PROGRAM GL9_Conveyor
VAR
	
	RUN_FWD_BIT_TO_EXIT : BOOL; // RUN FORWARD TO EXIT POSITION AFTER DROP
END_VAR
VAR // added by the converter: edge detectors and wires of the graphical bodies
    _w1 : BOOL;
END_VAR

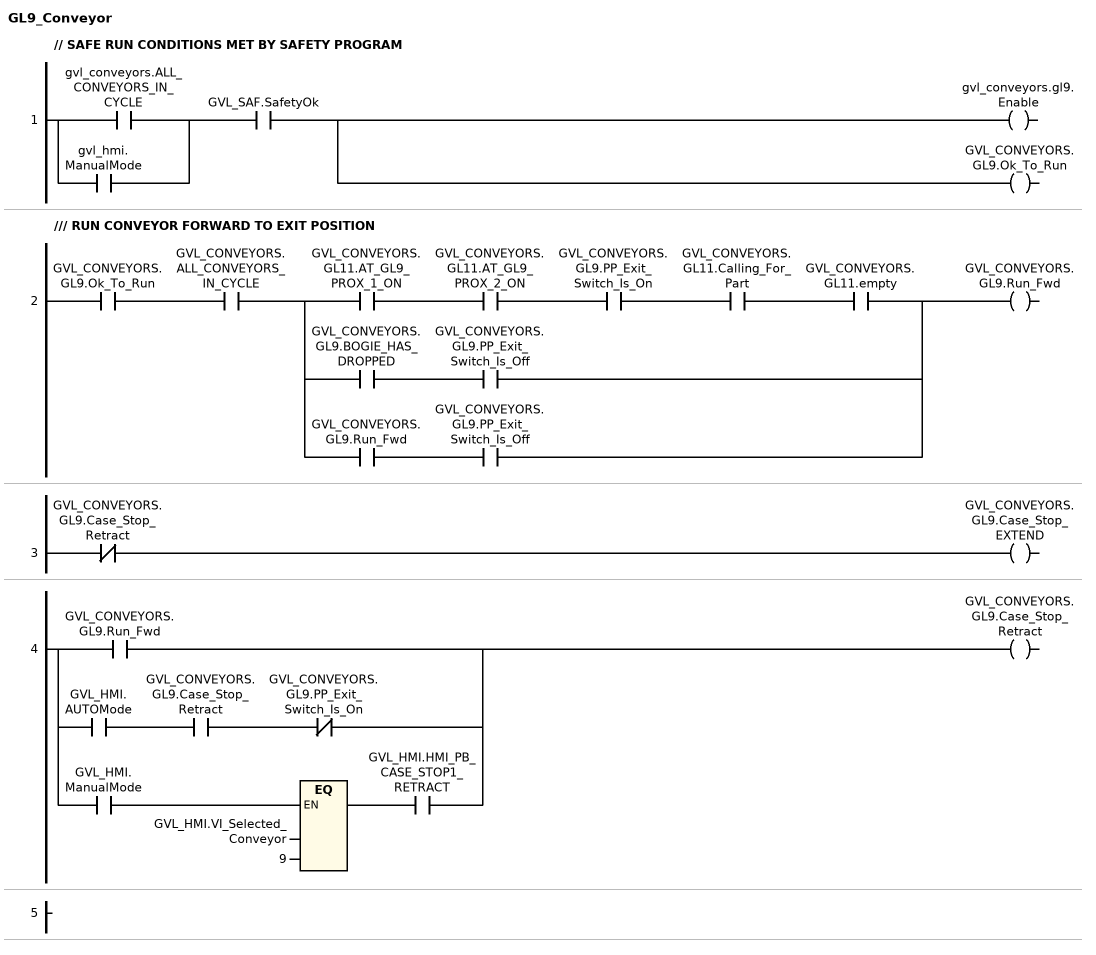
// NETWORK 1: // SAFE RUN CONDITIONS MET BY SAFETY PROGRAM
_w1 := (gvl_conveyors.ALL_CONVEYORS_IN_CYCLE OR gvl_hmi.ManualMode) AND GVL_SAF.SafetyOk;
gvl_conveyors.gl9.Enable := _w1;
GVL_CONVEYORS.GL9.Ok_To_Run := _w1;

// NETWORK 2: /// RUN CONVEYOR FORWARD TO EXIT POSITION
GVL_CONVEYORS.GL9.Run_Fwd := GVL_CONVEYORS.GL9.Ok_To_Run AND GVL_CONVEYORS.ALL_CONVEYORS_IN_CYCLE AND (GVL_CONVEYORS.GL11.AT_GL9_PROX_1_ON AND GVL_CONVEYORS.GL11.AT_GL9_PROX_2_ON AND GVL_CONVEYORS.GL9.PP_Exit_Switch_Is_On AND GVL_CONVEYORS.GL11.Calling_For_Part AND GVL_CONVEYORS.GL11.empty OR GVL_CONVEYORS.GL9.BOGIE_HAS_DROPPED AND GVL_CONVEYORS.GL9.PP_Exit_Switch_Is_Off OR GVL_CONVEYORS.GL9.Run_Fwd AND GVL_CONVEYORS.GL9.PP_Exit_Switch_Is_Off);

// NETWORK 3
GVL_CONVEYORS.GL9.Case_Stop_EXTEND := NOT GVL_CONVEYORS.GL9.Case_Stop_Retract;

// NETWORK 4
GVL_CONVEYORS.GL9.Case_Stop_Retract := GVL_CONVEYORS.GL9.Run_Fwd OR GVL_HMI.AUTOMode AND GVL_CONVEYORS.GL9.Case_Stop_Retract AND NOT GVL_CONVEYORS.GL9.PP_Exit_Switch_Is_On OR (GVL_HMI.ManualMode AND GVL_HMI.VI_Selected_Conveyor = 9) AND GVL_HMI.HMI_PB_CASE_STOP1_RETRACT;

// NETWORK 5

END_PROGRAM

(* stored: Version 1.1.0.1, ProductVersion 3.1.4024.12
   POU GL9_Conveyor: Id {5271b1d7-99d6-4485-887d-5b5142bcbef0}, SpecialFunc None *)
